# EPICS autosave request: ADApp/Db/PerkinElmer_settings.req
$(P)$(R)PEBadPixelFile
$(P)$(R)PECorrectionsDir
